// TIA Portal V16 export
// export: Created 2021-11-12T13:32:45.8227499Z, ExportSetting WithDefaults, DisplayName Totally Integrated Automation Portal, DisplayVersion V16 Update 3, DisplayName TIA Portal Version Control Interface, DisplayVersion V16 Update 2, DisplayName TIA Portal Openness, DisplayVersion V16 Update 3, DisplayName SINAMICS Startdrive Advanced, DisplayVersion V16 Update 5, DisplayName SINAMICS Startdrive G130, G150, S120, S150, SINAMICS MV, S210, DisplayVersion V16 Update 5, DisplayName SINAMICS Startdrive G110M, G120, G120C, G120D, G120P, G115D, DisplayVersion V16 Update 5, DisplayName STEP 7 Professional, DisplayVersion V16 Update 3, DisplayName STEP 7 Safety, DisplayVersion V16, DisplayName WinCC UA Professional, DisplayVersion V16 Update 3
DATA_BLOCK "IDB_StationBSN3"   // DB171
{ DB_Accessible_From_OPC_UA := 'FALSE' }
VERSION : 0.1
// stored: AutoNumber true, DBAccessibleFromOPCUA false, InstanceOfName StationBSN3, InstanceOfType FB
"StationBSN3"
   // VAR_INPUT
   //    IS_Inputs : "UDT_COMM_BSN3_CRS";
   // END_VAR
   // VAR_OUTPUT
   //    OS_Outputs : "UDT_COMM_CRS_BSN3";
   //    OS_Status : "UDT_BSN3_Status_specific";
   // END_VAR
   // VAR
   //    SF_TON_Tact : TON_TIME;
   //    SF_TON_1 { S7_SetPoint := 'True'} : TON_TIME;
   //    SF_Alarm1 : "STD_DI_Mon";
   //    SF_Alarm2 : "STD_DI_Mon";
   //    SF_Alarm3 : "STD_DI_Mon";
   //    SF_Alarm4 : "STD_DI_Mon";
   //    SF_Alarm5 : "STD_DI_Mon";
   //    SF_Alarm6 : "STD_DI_Mon";
   //    SF_Alarm7 : "STD_DI_Mon";
   //    SF_Alarm8 : "STD_DI_Mon";
   //    SF_CL01_Alarm { S7_SetPoint := 'True'} : "STD_DI_Mon";
   //    SF_CL01_Warning { S7_SetPoint := 'True'} : "STD_DI_Mon";
   //    SF_BoxPartCounter { S7_SetPoint := 'True'} : "STD_PartCounter";
   //    SS_Edge { S7_SetPoint := 'True'} : Array[0..15] of Bool;
   //    SS_ParamTemp : Struct
   //       PartType : Int;
   //       SPBurnerHigh : Int;
   //       SPTempSetpointZ1 : Int;
   //       SPTempSetpointZ2 : Int;
   //       SPTempSetpointZ3 : Int;
   //       SPTempSetpointZ4 : Int;
   //       SPTempSetpointZ5 : Int;
   //       SPTempSetpointZ6 : Int;
   //       SPTempSetpointZ7 : Int;
   //       ActPartTime : Int;
   //    END_STRUCT;
   //    SB1BoxExchangeReq { S7_SetPoint := 'True'} : Bool;
   //    SB1ReqBlockBeltMtion : Bool;
   //    SB1ReqBlockBeltMtion_Aux : Bool;
   //    SB1ParamChanged : Bool;
   //    ST_RunConv { S7_SetPoint := 'True'} : TOF_TIME;
   // END_VAR
BEGIN
END_DATA_BLOCK
